{attribute 'linkalways'} 
{attribute 'no_explicit_call' := 'This FB is a CLASS and must be accessed using methods or properties'}
{attribute 'enable_dynamic_creation'}
FUNCTION_BLOCK Node_F_VN_AppendToContainer_TcVnKeyPoint EXTENDS VisionNode
VAR
    stElement : _TcVnKeyPoint;
    ipContainer : _ITcVnContainer;
    hrPrev : _HRESULT(S_OK);
	hresult : _HRESULT(S_OK);
END_VAR

METHOD PUBLIC  Clone : I_Node
VAR
	pNode : POINTER TO Node_F_VN_AppendToContainer_TcVnKeyPoint;
END_VAR
pNode := __NEW(Node_F_VN_AppendToContainer_TcVnKeyPoint);
Clone := pNode^;
END_METHOD

METHOD FB_init : BOOL
VAR_INPUT
	bInitRetains : BOOL; // if TRUE, the retain variables are initialized (warm start / cold start)
	bInCopyCode : BOOL;  // if TRUE, the instance afterwards gets moved into the copy code (online change)
END_VAR
AddInput('stElement', stElement);
AddInput('ipContainer', ipContainer);
AddInput('hrPrev', hrPrev);
AddOutput('ipContainer', ipContainer);
AddOutput('hresult',hresult);
END_METHOD

METHOD PROTECTED OnExecute : HRESULT
hresult.Value := F_VN_AppendToContainer_TcVnKeyPoint(
    stElement := stElement.Value,
	ipContainer := ipContainer.Value,
	hrPrev:= hrPrev.Value);
END_METHOD

METHOD PUBLIC PreExecutionCheck
VAR_INPUT
	Check : I_PreExecutionChecks;
END_VAR
Check.IsTrue(ipContainer.IsValid, 'ipContainer must be a valid container');
END_METHOD

END_FUNCTION_BLOCK

(* stored: Version 1.1.0.1, ProductVersion 3.1.4024.13
   POU Node_F_VN_AppendToContainer_TcVnKeyPoint: Id {fdaad668-ed25-4da8-b0b7-5a6086e33e19}, SpecialFunc None
   Folder Constructor: Id {5e809133-e508-4e8c-828a-b756fc28d5c8}
   Method Clone: Id {051ef1dd-38bf-4a89-9f4b-a9294db47c91}
   Method FB_init: Id {206bcd3f-6825-4b86-8363-919a6b32276a}
   Method OnExecute: Id {78b0683c-bd02-4263-8532-3054dd7d2ba2}
   Method PreExecutionCheck: Id {39eaea13-b410-49f3-9b2b-9f5f38e3d3f3} *)
